FUNCTION_BLOCK FB_MotorSS
VAR_INPUT
	mxReset							: BOOL;
	mxEmergency						: BOOL;
	mxAutoMode						: BOOL;
	mxDisableManualAutoTrigger		: BOOL := FALSE; // If this bit is enabled, the outputs status is not changed when change from/to automode happens
END_VAR
VAR_OUTPUT
(*Errors*)
	Errors							: ST_MotorSSErrors;
	mxErrorInit						: BOOL;		(* Error, stop immediately. Initialisation neccesary *)
	mxErrorStopinPos				: BOOL;		(* Error, stop in position. Only reset neccesary *)

(* State vars *)
	mxCycleBusy						: BOOL;
	mxInitBusy						: BOOL;
	
(* Vars *)
	mxInitialized					: BOOL;
	IsRunning						: BOOL;
	
END_VAR
VAR
	ixSSFailure						AT %I* : BOOL;
	ixMaintenance					AT %I* : BOOL;
	ixIsRunning						AT %I* : BOOL;
	Q								AT %Q* : BOOL;
	
	Hmi_On							: BOOL;
	RT_AutoMode						: R_TRIG;
	SR_ErrorMaintenance				: SR;
	SR_ErrorSS: SR;
	mxTest: BOOL;
END_VAR

Error();

(* Reset hmi when switched to automode*)
RT_AutoMode(CLK:= mxAutoMode);

// if manual mode becomes active, the manualmode (hmi) is over written by its current state.
// this ensures that the motor keeps running when it was running and is switched to manual. 
IF RT_AutoMode.Q AND NOT mxDisableManualAutoTrigger THEN Hmi_On:= Q; END_IF	

(* Manual control *)
//IF NOT mxAutoMode THEN Q:= Hmi_On; END_IF

IsRunning:= ixIsRunning;

ACTION Error:
SR_ErrorSS(SET1:= NOT ixSSFailure, RESET:= mxReset, Q1=> Errors.SofstarterFailure);
SR_ErrorMaintenance(SET1:= NOT ixMaintenance, RESET:= mxReset, Q1=> Errors.Maintenance);

(******************************************************************************************************)
mxErrorStopinPos:= FALSE;
mxErrorInit:= Errors.SofstarterFailure OR Errors.Maintenance;
END_ACTION

METHOD M_Init

Q:= FALSE;
END_METHOD

METHOD M_Start : BOOL
VAR_INPUT
END_VAR
Q:=TRUE;

(* Return Value *)
M_Start:= Q;
END_METHOD

METHOD M_Stop : BOOL
VAR_INPUT
END_VAR
Q:= FALSE;

(* Return Value *)
M_Stop:= NOT Q;
END_METHOD

END_FUNCTION_BLOCK

(* stored: Version 1.1.0.1, ProductVersion 3.1.4020.12
   POU FB_MotorSS: Id {0f3f7470-7033-406e-bdbd-25eedababbe4}, SpecialFunc None
   Action Error: Id {d3b05e4f-983f-4ce1-9d01-5d763a3b0874}
   Method M_Init: Id {8177ab19-9c29-427f-9536-cabb418bdd60}
   Method M_Start: Id {ead3873f-3efc-4d3d-9e8c-cb022a34ac7c}
   Method M_Stop: Id {a7c6335d-e6a2-4c35-82e3-b5d76c4d265e} *)
